FUNCTION_BLOCK POU2
VAR_INPUT
END_VAR
VAR_OUTPUT
END_VAR
VAR
END_VAR

END_FUNCTION_BLOCK

(* stored: Version 1.1.0.1, ProductVersion 3.1.4020.12
   POU POU2: Id {00b92a5b-c033-4c7c-87be-80a19caec9da}, SpecialFunc None *)
